# EPICS autosave request: ADApp/Db/NDCircularBuff_settings.req
$(P)$(R)TriggerA
$(P)$(R)TriggerB
$(P)$(R)TriggerCalc
$(P)$(R)PRECOUNT
$(P)$(R)POSTCOUNT
$(P)$(R)ReArm
